FUNCTION_BLOCK FB_NcAxis
VAR CONSTANT

	sPosBiasStateTextDef: ARRAY[0..2] OF STRING:=	['State 0: Wait for Start',
										'State 1: Read Pos Bias, calculate new Pos Bias',
										'State 2: Write Pos Bias'];

	tPosBiasStateTimeouts: ARRAY[0..2] OF TIME:=  [T#10S, T#10S, T#10S];
	
END_VAR
VAR_INPUT
	mxEnable						: BOOL;
	mxInhibit						: BOOL :=TRUE;
	mxAutoMode						: BOOL;
	mxReset							: BOOL;
	mxFirstCycle					: BOOL;
	mxEmergency						: BOOL;
	mxSimulation					: BOOL;
	mxResetCycle					: BOOL;
	mxDisable_Positive				: BOOL; 
	mxDisable_Negative				: BOOL;
	mxBlockHMI						: BOOL:= FALSE;
	mrOverride						: LREAL;
	mrVelocityManual				: LREAL;
	mxResetPosBiasState				: BOOL;
	mxZeroCommand					: BOOL;
	mrHomePos						: LREAL;
END_VAR
VAR_IN_OUT
	SysParameters					: ST_NcAxis_SysPar;
END_VAR
VAR_OUTPUT
	mxCycleBusy						: BOOL;
	mxRunning						: BOOL;
	mxAxisIsMoving					: BOOL;
	///Errors
	Errors							: st_NcAxis_Errors;
	Error							: BOOL;
	ErrorStop						: BOOL;

	axStatus						:ST_AxisStatus;
	ActPosition						:LREAL;
	ActVelocity						:LREAL;

	axAxis							: AXIS_REF;

	mxPosBiasBusy					: BOOL;
	mxPosBiasHasError				: BOOL;
	SignalLightStatus					: BOOL;(* Needed in the HMI, for changing the color of the signal light *)	
END_VAR
VAR
	HmiStatus: UINT;
	HmiControl: UINT;
	HMI_ReadEncoder:BOOL;
	HMI_ReadmInc:LREAL;
	HMI_WriteEncoder:BOOL;
	HMI_WritemInc: LREAL;
	
	HMI_Forward				: BOOL;
	HMI_Backward			: BOOL;
	mxActivateAuto:BOOL;
	mxActivateManual:BOOL;
	mxActivated:BOOL;
	
	MCPower							: MC_Power;
	MCReset							: MC_Reset;
	MCJog							: MC_Jog;
	MCStop							: MC_Stop;
	MCHome							: MC_Home;
	MCMoveAbsolute					: ARRAY[0..1] OF MC_MoveAbsolute;
	mxMoveAbsNr						: INT;
	MCMoveVelocity					: ARRAY[0..1] OF MC_MoveVelocity;
	mxMoveVelocityNr				: INT;	
	MCReadParameter					: MC_ReadParameter;
	MCReadAxisError					: MC_ReadAxisError;
	MCWriteParameter				: MC_WriteParameter; 
 	MCSetPosition					: MC_SetPosition;
	MCReadStatus					: MC_ReadStatus;
	mcResetDrive					: FB_SoEReset_ByDriveRef;
	iDriveRef						AT %I* :ST_PLCDriveRef;
	
(*Drive parameters*)	
	mcBlendingMode					: MC_BufferMode;

	miState							: INT	:=0;
	miStopState						: INT	:=0;
	miOldstate						: INT	:=0;
	mxTransitionState				: BOOL	:= FALSE;
	sStateText						: STRING;	
	
 	exPosBiasTimeOut				: BOOL;		(* Timeout for the whole programcycle *)
	miPosBiasState					: INT	:=0;
	miPosBiasOldstate				: INT	:=0;
	mxPosBiasTransitionState		: BOOL	:= FALSE;
	sPosBiasStateText				: STRING;
	PosBiasTimeout					: TON;

(* Vars *)
	mxPosBiasTimeoutEnable			: BOOL;
	PosBiasTime						: REAL;

	mrStoredAxisPosition			: LREAL;
	mxPositionError					: BOOL;

	AdsReadPosBias					: ADSREAD;
	AdsWritePosBias					: ADSWRITE;

	PositionBiasRead 				: LREAL;
	
	(* Errors *)
	SR_DrivePower					: SR;
	SR_DriveJog						: SR;
	SR_DriveStatus					: SR;
	SR_DriveStop					: SR;
	SR_DriveReset					: SR;
	SR_Home							: SR;
	SR_Restart						: SR;
	SR_MotorError					: SR;
	SR_DriveAbsError				: SR;
	SR_DriveVelocity				: SR;
	SR_WriteParameter				: SR;
	SR_ReadParameter				: SR;
	SR_LagError						: SR;
 
	x: INT;
	
	mxCycleHasError					: BOOL;
	
(*Timers*)
	T_Power_On						: TON;
	T_Power_Off						: TOF;
	CycleTimeout					: TON;

(*Raising Edge detections*)
	RT_AutoManual					: R_TRIG;
	FT_AutoManual					: F_TRIG;
	RT_AutoManualHMI				: R_TRIG;
	CycleTimeOutUpFlank				: R_TRIG;
	PosBiasTimeOutUpFlank			: R_TRIG;

(* Vars *)
	mxCycleTimeoutEnable			: BOOL;
	CycleTime						: REAL;
	SR_CycleTimeOut					: SR;	
	mrPosition: LREAL;
	mrCheckPosition: LREAL;
	mxMoveForw: BOOL;
	mxSimulationDO	:INT:=0;	(*0= direct onposition, 1=seconds OnPosition, 2=not on position first and second*)
	ErrorIDMoveAbs1: UDINT;
	ErrorIDMoveAbs0: UDINT;

	T_Delay: TON;
	T_StandstillDelay: TON;
	miReadErrorID: DWORD;
	miReadAxisErrorID: DWORD;
END_VAR

Alarms();
WritePosBias();
HMI();
DriveActions();

ACTION Alarms:
SR_DrivePower(SET1:=MCPower.Error , RESET:=mxReset , Q1=> errors.exDrivePower);
SR_DriveJog(SET1:= MCJog.Error, RESET:=mxReset , Q1=> errors.exDriveJog);
SR_DriveStatus(SET1:= axAxis.Status.Error, RESET:=mxReset , Q1=> errors.exDriveStatus);
SR_DriveReset(SET1:= MCReset.Error, RESET:= mxReset, Q1=>errors.exDriveReset );
SR_DriveAbsError(SET1:=MCMoveAbsolute[0].Error OR MCMoveAbsolute[1].Error, RESET:= mxReset, Q1=>errors.exDriveAbsoluut );
SR_DriveStop(SET1:= MCStop.Error, RESET:= mxReset, Q1=>errors.exDriveStop );
SR_WriteParameter(SET1:= MCWriteParameter.Error, RESET:= mxReset, Q1=>errors.exWriteParameter );
SR_ReadParameter(SET1:= MCReadParameter.Error, RESET:= mxReset, Q1=>errors.exReadParameter );
SR_Home(SET1:= MCHome.Error, RESET:= mxReset, Q1=>errors.exHome );
SR_DriveVelocity(SET1:= MCMoveVelocity[0].Error OR MCMoveVelocity[0].Error, RESET:= mxReset, Q1=> Errors.exDriveVelocity);
SR_LagError(SET1:=(MCMoveAbsolute[0].ErrorID = 17744 AND MCMoveAbsolute[0].Error) OR 
						 (MCMoveAbsolute[1].ErrorID = 17744 AND MCMoveAbsolute[1].Error) OR
						 (MCJog.ErrorID = 17744 AND MCJog.Error) OR 
						 (MCMoveVelocity[0].ErrorID = 17744 AND MCMoveVelocity[0].Error) OR 
						 (MCMoveVelocity[1].ErrorID = 17744 AND MCMoveVelocity[1].Error) OR
						 axStatus.ErrorID = 17744
						 , RESET:= mxReset, Q1=>errors.exLagError );

ErrorStop:= errors.exLagError OR errors.exWriteParameter OR errors.exReadParameter OR 
	errors.exDriveStop OR errors.exDrivePower OR errors.exDriveJog  OR  errors.exDriveStatus OR 
	errors.exDriveReset OR Errors.exDriveAbsoluut OR Errors.exDriveVelocity OR errors.exHome;
END_ACTION

ACTION DriveActions:
(*read axis status*)
axAxis.ReadStatus();
axStatus:= axAxis.Status;
ActPosition:=axAxis.NcToPlc.ActPos;
ActVelocity:=axAxis.NcToPlc.ActVelo;
mxAxisIsMoving:= axAxis.Status.Moving;

	(*Power Axis*)
T_Power_On(IN:=(NOT mxInhibit), PT:= T#10MS);
T_Power_Off(IN:=T_Power_On.Q , PT:=T#5S , Q=> , ET=> );
(*power axis*)	
MCPower(
	Axis:= axAxis, 
	Enable:=NOT mxEmergency AND (T_Power_On.Q OR T_Power_Off.Q),  
	Enable_Positive:= NOT mxDisable_Positive , 
	Enable_Negative:= NOT mxDisable_Negative , 
	Override:=, 
	BufferMode:= , 
	Options:= , 
	Status=> , 
	Busy=> , 
	Active=> , 
	Error=> , 
	ErrorID=> );
	 
(*Drive run action manual*)
MCJog(
	Axis:= axAxis, 
	JogForward:= ,
	JogBackwards:= ,
	Mode:=MC_JOGMODE_CONTINOUS , 
	Position:= , 
	Velocity:= mrVelocityManual, 
	Acceleration:= , 
	Deceleration:= , 
	Jerk:= , 
	Done=> , 
	Busy=> , 
	Active=> , 
	CommandAborted=> , 
	Error=> , 
	ErrorID=> );
	MCJog.JogForward:=FALSE; 	
	MCJog.JogBackwards:=FALSE;

(*Drive Reset*)
MCReset(
	Axis:=axAxis , 
	Execute:=(mxReset AND (axAxis.Status.Error OR Error)), 
	Done=> , 
	Busy=> , 
	Error=> , 
	ErrorID=> );

	(*Reset*)
//DriveAxis.mcReset(Execute:= mxReset AND DriveAxis.mcStatus.Error, Axis:= axAxis);

(* Reset Drive Error *)
mcResetDrive.stDriveRef.sNetId:= F_CreateAmsNetId(iDriveRef.aNetId);
mcResetDrive.stDriveRef.nSlaveAddr:= iDriveRef.nSlaveAddr;
mcResetDrive.stDriveRef.nDriveNo:= iDriveRef.nDriveNo;


mcResetDrive(
	bExecute:= mxReset AND axAxis.Status.DriveDeviceError,
	tTimeout:= t#10s);
	
(*Move absolute fb 1*) 
	MCMoveAbsolute[0](
			Axis:= axAxis, 
			Execute:=, 
			Position:= , 
			Velocity:= , 
			Acceleration:= , 
			Deceleration:= , 
			Jerk:= , 
			BufferMode:= , 
			Options:= , 
			Done=> , 
			Busy=> , 
			Active=> , 
			CommandAborted=> , 
			Error=> , 
			ErrorID=> );
MCMoveAbsolute[0].Execute:=FALSE;
IF MCMoveAbsolute[0].ErrorID > 0 THEN ErrorIDMoveAbs0:=MCMoveAbsolute[0].ErrorID; END_IF;
(*Move absolute fb 2*)
	MCMoveAbsolute[1](
			Axis:= axAxis, 
			Execute:=, 
			Position:= , 
			Velocity:= , 
			Acceleration:= , 
			Deceleration:= , 
			Jerk:= , 
			BufferMode:=, 
			Options:= , 
			Done=> , 
			Busy=> , 
			Active=> , 
			CommandAborted=> , 
			Error=> , 
			ErrorID=>ErrorIDMoveAbs1 );
MCMoveAbsolute[1].Execute:=FALSE;
IF MCMoveAbsolute[1].ErrorID > 0 THEN ErrorIDMoveAbs0:=MCMoveAbsolute[1].ErrorID; END_IF;
(*Move velocity fb 1*)
MCMoveVelocity[0](
	Axis:=axAxis , 
	Execute:= , 
	Velocity:= , 
	Acceleration:= , 
	Deceleration:= , 
	Jerk:= , 
	Direction:= , 
	BufferMode:= , 
	Options:= , 
	InVelocity=> , 
	Busy=> , 
	Active=> , 
	CommandAborted=> , 
	Error=> , 
	ErrorID=> );
			
MCMoveVelocity[0].Execute:=FALSE;		
 (*Move velocity fb 2*)
MCMoveVelocity[1](
	Axis:=axAxis , 
	Execute:= , 
	Velocity:= , 
	Acceleration:= , 
	Deceleration:= , 
	Jerk:= , 
	Direction:= , 
	BufferMode:= , 
	Options:= , 
	InVelocity=> , 
	Busy=> , 
	Active=> , 
	CommandAborted=> , 
	Error=> , 
	ErrorID=> );
			
MCMoveVelocity[1].Execute:=FALSE;		

MCStop(
	Axis:=axAxis , 
	Execute:= , 
	Deceleration:= , 
	Jerk:= , 
	Options:= , 
	Done=> , 
	Busy=> , 
	Active=> , 
	CommandAborted=> , 
	Error=> , 
	ErrorID=> );
MCStop.Execute:=FALSE;

(*Homing*)
MCHome(
	Axis:=axAxis , 
	Execute:= , 
	Position:=  , 
	HomingMode:=  , 
	BufferMode:= , 
	Options:= , 
	bCalibrationCam:= , 
	Done=> , 
	Busy=> , 
	Active=> , 
	CommandAborted=> , 
	Error=> , 
	ErrorID=> );
MCHome.Execute:=FALSE;
	
(*Read a parameter*)
MCReadParameter(
	Axis:=axAxis , 
	Enable:= , 
	ParameterNumber:= , 
	ReadMode:=E_ReadMode.READMODE_CYCLIC , 
	Valid=> , 
	Busy=> , 
	Error=> , 
	ErrorID=> , 
	Value=> );
MCReadParameter.Enable:=FALSE;

(*Write a parameter*)	
MCWriteParameter(
	Axis:= axAxis, 
	Execute:= , 
	ParameterNumber:= , 
	Value:= , 
	Done=> , 
	Busy=> , 
	Error=> , 
	ErrorID=> );
MCWriteParameter.Execute:=FALSE;

MCSetPosition(
	Axis:= axAxis, 
	Execute:= , 
	Position:= , 
	Mode:=FALSE , 
	Options:= , 
	Done=> , 
	Busy=> , 
	Error=> , 
	ErrorID=> );
	MCSetPosition.Execute:=FALSE;	

MCReadAxisError(
	Axis:=axAxis , 
	Enable:=TRUE , 
	Valid=> , 
	Busy=> , 
	Error=> , 
	ErrorID=> miReadErrorID, 
	AxisErrorID=>miReadAxisErrorID );
	(*
MCReadStatus(
	Axis:= axAxis, 
	Enable:= , 
	Valid=> , 
	Busy=> , 
	Error=> , 
	ErrorID=> , 
	ErrorStop=> , 
	Disabled=> , 
	Stopping=> , 
	StandStill=> , 
	DiscreteMotion=> , 
	ContinuousMotion=> , 
	SynchronizedMotion=> , 
	Homing=> , 
	ConstantVelocity=> , 
	Accelerating=> , 
	Decelerating=> , 
	Status=> );*)
END_ACTION

ACTION HMI:
(*Read ax encoder parameter minc*)
IF HMI_ReadEncoder THEN
	HMI_ReadmInc :=	M_ReadParameter(MC_AxisParameter.AxisEncoderScalingFactor);
END_IF
(*Write ax encoder parameter*)
IF HMI_WriteEncoder THEN
	M_WriteParameter(miParameterNr:=MC_AxisParameter.AxisEncoderScalingFactor , miValue:= HMI_WritemInc );
END_IF

IF mxAutoMode THEN
	MCPower.Override:=mrOverride;
ELSE
	MCPower.Override:=mrOverride(*parameters.VelocityManual*);		
END_IF;

RT_AutoManual(CLK:= mxAutoMode);
FT_AutoManual(CLK:= mxAutoMode);

(*Set output*)
mxActivateAuto:= (mxEnable AND mxAutomode);
mxActivateManual := (mxEnable AND NOT mxAutoMode);

IF HMI_Forward AND axAxis.Status.Operational AND NOT SR_Restart.Q1 AND T_Power_On.Q AND NOT mxAutomode THEN
	MCJog.JogForward := TRUE ;
	MCJog.Velocity:= mrVelocityManual;
END_IF
IF HMI_Backward AND axAxis.Status.Operational AND NOT SR_Restart.Q1 AND T_Power_On.Q AND NOT mxAutoMode THEN
	MCJog.JogBackwards :=TRUE;
	MCJog.Velocity:= mrVelocityManual;
END_IF
END_ACTION

METHOD M_Home : BOOL;
VAR_INPUT
	mrHomePosition		: LREAL;
	MCMode				: MC_HomingMode;
END_VAR
McHome.Position:= mrHomePosition;
McHome.HomingMode:= MCMode;

McHome.Execute:= TRUE;


(* Return Value *)
M_Home:=MCHome.Done;
END_METHOD

METHOD M_MoveAbsolute : BOOL
VAR_INPUT
	Velocity				:LREAL;			
	Position				:LREAL;
END_VAR
(*compare for different setpoints, if so change fb mcMoveAbsolute*)
IF 	(MCMoveAbsolute[mxMoveAbsNr].Position <> Position) OR 
	(MCMoveAbsolute[mxMoveAbsNr].Velocity <> Velocity) THEN

	IF mxMoveAbsNr = 0 THEN
		mxMoveAbsNr :=1;
	ELSE
		mxMoveAbsNr :=0;
	END_IF
	
	(*Write parameters*)
	MCMoveAbsolute[mxMoveAbsNr].Position:=Position;
	MCMoveAbsolute[mxMoveAbsNr].Velocity:=Velocity;
(*	IF Velocity > 0.0 	THEN  MCMoveAbsolute[mxMoveAbsNr].Velocity:=Velocity; 		 ELSE MCMoveAbsolute[mxMoveAbsNr].Velocity:=parameters.VelocityAuto; 	END_IF*) 
END_IF

MCMoveAbsolute[mxMoveAbsNr].Execute:=TRUE;

(* Return value *)
M_MoveAbsolute:=MCMoveAbsolute[mxMoveAbsNr].Done;
END_METHOD

METHOD M_MoveVelocity : BOOL
VAR_INPUT
	Velocity			: LREAL;			
	Direction			: MC_Direction;
END_VAR
(*compare for different setpoints, if so change fb mcMoveVelocity*)
IF 	(MCMoveVelocity[mxMoveVelocityNr].Velocity <> Velocity) THEN

	IF mxMoveVelocityNr = 0 THEN
		mxMoveVelocityNr :=1;
	ELSE
		mxMoveVelocityNr :=0;
	END_IF

	(*Write parameters*)
	MCMoveVelocity[mxMoveAbsNr].Velocity:=Velocity;
(*	IF Velocity > 0 	THEN MCMoveVelocity[mxMoveVelocityNr].Velocity:=Velocity; 			ELSE MCMoveVelocity[mxMoveVelocityNr].Velocity:=parameters.VelocityAuto; 		END_IF*)

END_IF

MCMoveVelocity[mxMoveVelocityNr].Execute:=TRUE;
MCMoveVelocity[mxMoveVelocityNr].Direction:=Direction;

(*Give return value*)
M_MoveVelocity:=MCMoveVelocity[mxMoveVelocityNr].Active;
END_METHOD

METHOD M_ReadParameter : LREAL
VAR_INPUT
		miParameterNr:INT;
END_VAR
MCReadParameter.ParameterNumber:=miParameterNr;
MCReadParameter.Enable:=TRUE;

M_ReadParameter:=MCReadParameter.Value;
END_METHOD

METHOD M_Reset : BOOL
VAR_INPUT
	
END_VAR

(* Return Value *)
M_Reset:= MCReset.Done;
END_METHOD

METHOD M_SetPosition : BOOL
VAR_INPUT
	NewPosition:LREAL;
END_VAR
MCSetPosition.Position:=NewPosition;
MCSetPosition.Execute:=TRUE;

M_SetPosition:=MCSetPosition.Done;
END_METHOD

METHOD M_Stop : BOOL
MCStop.Execute:=TRUE;

(* Return Value *)
M_Stop:= MCStop.Done;
END_METHOD

METHOD M_WriteParameter : BOOL
VAR_INPUT
	miParameterNr:INT;
	miValue:LREAL;
END_VAR
MCWriteParameter.ParameterNumber:=miParameterNr;
MCWriteParameter.Value:=miValue;
MCWriteParameter.Execute:=TRUE;

M_WriteParameter:=MCWriteParameter.Done;
END_METHOD

ACTION WritePosBias:
(*StateChange (Transition)  Signalgeneration*)
mxPosBiasTransitionState:=(miPosBiasState<>miPosBiasOldstate);
(*State text*)
sPosBiasStateText:=sPosBiasStateTextDef[miPosBiasState];
(*Timeout Watchdog for Statemachine*)
mxPosBiasTimeoutEnable:=NOT (miPosBiasState=0)  AND NOT mxReset;

PosBiasTimeout(IN:=mxPosBiasTimeoutEnable  , PT:=tPosBiasStateTimeouts[miPosBiasState] );
PosBiasTimeOutUpFlank(CLK:=PosBiasTimeout.Q );
miPosBiasOldstate:=miPosBiasState;

(*Set Errorbit when Raising edge of Timeout has been detected*)
IF PosBiasTimeOutUpFlank.Q THEN
	exPosBiasTimeOut:=TRUE; 			(* 1 Timeout for the whole programcycle *)
END_IF

(*Function to reset the Statemachine*)
IF mxResetPosBiasState THEN
	mxResetPosBiasState:=FALSE;
	miPosBiasState:=0;
	miPosBiasOldstate:=miPosBiasState;
	mxPosBiasTransitionState:=FALSE;

	AdsReadPosBias.READ:= FALSE;
	AdsWritePosBias.WRITE:= FALSE;

	mxZeroCommand:= FALSE;
	SignalLightStatus:= FALSE;
END_IF

AdsReadPosBias(
	NETID:= '',
	PORT:= 500,
	IDXGRP:= SysParameters.IDXGRP,
	IDXOFFS:= 16#7,
	LEN:= 8,
	DESTADDR:= ADR(PositionBiasRead),
	TMOUT:= T#1s);

AdsWritePosBias(
	NETID:= '',
	PORT:= 500,
	IDXGRP:= SysParameters.IDXGRP,
	IDXOFFS:= 16#7,
	LEN:= 8,
	SRCADDR:= ADR(SysParameters.PositionBias),
	TMOUT:= T#1s);

(*Definition State has Error*)
mxPosBiasHasError:=FALSE;

(*Cycle State's*)
CASE miPosBiasState OF
	(*Wait for Start *)
	0:
		(* Zero command from HMI *)
		IF mxZeroCommand THEN
			mxZeroCommand:= FALSE;
			SignalLightStatus:= FALSE;

			AdsReadPosBias.READ:= TRUE;
			miPosBiasState:= 1;
		END_IF

		(* PLC startup *)
		IF mxFirstCycle THEN
			SignalLightStatus:= FALSE;

			AdsWritePosBias.WRITE:= TRUE;
			miPosBiasState:= 2;
		END_IF

	(* Calculate new Position Bias with actual bias and act position *)
	1:
		IF NOT AdsReadPosBias.BUSY THEN
			AdsReadPosBias.READ:= FALSE;

			SysParameters.PositionBias:= mrHomePos - axAxis.NcToPlc.ActPos + PositionBiasRead;
			AdsWritePosBias.WRITE:= TRUE;

			miPosBiasState:= 2;
		END_IF

	(* Write new position bias *)
	2:
		IF NOT AdsWritePosBias.BUSY THEN
			AdsWritePosBias.WRITE:= FALSE;
			SignalLightStatus:= TRUE;

			miPosBiasState:= 0;
		END_IF
END_CASE

(*Set Busy bit FOR Statemachine*)
mxPosBiasBusy:=(miposBiasState<>0);
END_ACTION

END_FUNCTION_BLOCK

(* stored: Version 1.1.0.1, ProductVersion 3.1.4020.12
   POU FB_NcAxis: Id {aa5a62ae-161e-4de1-ab36-80c9a7694333}, SpecialFunc None
   Action Alarms: Id {f58ab993-5ae0-463b-aeab-0073f58ca206}
   Action DriveActions: Id {224c1903-023a-4ee2-8320-b68027136e41}
   Action HMI: Id {eb8fabfc-d4e1-4347-858a-5a775d72ba78}
   Method M_Home: Id {bc90398b-d2be-47ef-b133-5c702c2e92ab}
   Method M_MoveAbsolute: Id {a80ceb5a-497b-4f0a-9a7f-3af21bbe59cf}
   Method M_MoveVelocity: Id {75e5abaf-82f2-4bb9-8aec-abdd0b3b7e72}
   Method M_ReadParameter: Id {a3ec4172-9efd-401e-949e-d2288dfad79c}
   Method M_Reset: Id {f5452be7-27f7-4379-9f0b-026febb0f92e}
   Method M_SetPosition: Id {d7bf1ce8-11e0-42f8-822d-d2b5c6779695}
   Method M_Stop: Id {de26110d-985c-4a8a-8e4f-0907dc3050a3}
   Method M_WriteParameter: Id {f64eec33-ed5c-4233-8efd-e2c86928db68}
   Action WritePosBias: Id {022419e5-638a-462e-a879-1fd64df2c80e} *)
